{attribute addProperty BoxType "EL3602-0000-0016"}
{attribute addProperty Id "AI_Inputs_ChannelAT %I*ARRAY[0..1] OF AI_Inputs_Channel_513C0694176220WcStateAT %I*WcState_F855686C1620InfoDataAT %I*InfoData_BC63D37F80100"}
{attribute addProperty CRC "1779321452"}
{attribute addProperty SizeInBites "272"}
{attribute addProperty SizeInBytes "34"}
TYPE EL3602_9C69A51A :
STRUCT
	{attribute addProperty Name "AI_Inputs_Channel"}
	AI_Inputs_Channel : ARRAY[0..1] OF AI_Inputs_Channel_513C0694;
	{attribute addProperty Name "WcState"}
	WcState : WcState_F855686C;
	{attribute addProperty Name "InfoData"}
	InfoData : InfoData_BC63D37F;
END_STRUCT
END_TYPE

(* stored: Version 1.2.0.0, ProductVersion 3.1.4024.9
   DUT EL3602_9C69A51A: Id {32178f7f-3231-4e42-ba45-d6ea03628b75} *)
